FUNCTION F_ComputeTagSize : UDINT
VAR_INPUT
    nFieldnumber    : UDINT;
END_VAR


F_ComputeTagSize := F_ComputeRawVarint32Size(nValue:= F_MakeTag(nFieldNumber, 0));

END_FUNCTION

(* stored: Version 1.1.0.1
   POU F_ComputeTagSize: Id {66d0678b-c751-4a1c-904a-a7ec1e3eed3b}, SpecialFunc None *)
